(*
  Detects Marks and generates StartTrigger based on one EL1252 timestamp input I/O.
  Implements a CameraTrigger instance as well.
  
  Additionally:
    - returns lateral offset (+/- in [m]) to center of detected marks.
    - manages & supervises mark sequence
    - is a CameraTrigger as well
    - supports simulation mode
  
  NOTE: 
    - a mark has always a rising and falling edge of the sensor (triangle)
    - center position is the middle of the triangular mark

*)
FUNCTION_BLOCK FB_MarkDetection_v1 EXTENDS T_NamedBase IMPLEMENTS I_StartPosDetect, I_CameraTrigger, I_Sim
VAR_INPUT
  (*EL1252*)
  bIKp_StartSensor          AT%I* : BOOL;             (*Sensor start trigger*)
  tIKp_TimeStampPos         AT%I* : T_DCTIME64;       (*TimeStamp Pos_Edge @EL1252*)
  tIKn_TimeStampNeg         AT%I* : T_DCTIME64;       (*TimeStamp Neg_Edge @EL1252*)

  // configuration
  bEnable                         : BOOL;             (*Enable start pos detection sensor (from extern)*)
  bAutomaticMode                  : BOOL;             (*machine is in automatic mode *)
  nCurrentPos                     : DINT;             (*current position in Pulses/Subpixels*)
  fCurrentSpeed                   : LREAL;            (*actual speed of conveyor in [m/s]*)
  bReverse                        : BOOL;             (*reverse printing same roll feeded in opposite direction, check falling edge in this case*)
  
  // Debug & Test
  bManualTrigger                  : BOOL;             // Manual start trigger
  bManualReset                    : BOOL;             // Manaul reset detection
END_VAR
VAR
  bInitOk                         : BOOL;             // fb initialized

  // config
  _fResolution                    : LREAL := 1;       // current used print resolution (dpi*SubPx)
  _pFbMarkDefinition              : POINTER TO FB_MarkDefinition;      // mark definition
  _iCamera                        : I_Camera;         // camera interface
  // settings                                    
  _bUseCameraTrigger              : BOOL;             // (cam specific setting) Generate camera trigger output
  _bUseCameraTriggerFeedback      : BOOL;             // (cam specific setting) Evaluate camera triggered feedback
  _bCamManualTeachMode            : BOOL;             // cam in manual teach mode
  _fSubstrateLength               : LREAL;            // Substrate length in [m] (should be repeat ength)
  _fTriggerDistance               : LREAL;            // Distance between Sensor and Trigger [m]
  _fTriggerLength                 : LREAL := 10;      // Length of trigger signal in ms, min. 3 bus cycles
  _iActiveCam                     : I_CameraTriggerDevice;  // active camera interface (set by Enable() on I_CameraTrigger)

  // sensor
  bSheetActive                    : BOOL;             (*sheet is scanning*)
  bSpeedValid                     : BOOL;             (*speed is valid*)
  bTriggerArmed                   : BOOL;             (*trigger is armed*)
  bCamValid                       : BOOL;             (*camera is valid*)
  bMarkValid                      : BOOL;             (*definition is valid marks&substrate*)
  
  // helper
  rfT_Enable                      : RF_TRIG;          // edge detection enable
  bResetDetection                 : BOOL;             // Reset request for checkForMark() internals
  isStartMark                     : BOOL;
  isMarkError                     : BOOL;
  nMarkSelection                  : UDINT := 1;       // Current selected mask to search
  pMarkSearch                     : POINTER TO ST_MarkDefinition;
  _fSubstrateLengthEffective      : LREAL;            // Substrate length in [m]
  
  // time calculations
  tNowDc                          : T_DCTIME64;       // Get Current Timestamp (now)
  fCycleTime                      : LREAL;            // Current calculated cycle time [s]
  
  // I_StartPosDetect
  _bStartTrig                     : BOOL;             // Start Trigger Edge
  _nX0                            : DINT;             // X0 Position [SubPx]
  _bValid                         : BOOL;             //
  
  // simulation & debug
  _bSimEnable                     : BOOL;             // simulation mode enabled
  _bVerbose                       : BOOL;             // verbose mode
  _fSubstrateGap                  : LREAL;            // Gap between two substrates (sheets/repeats) for simulation
  
  // local for checkForMark
  rfEdgeSensor                    : RF_TRIG;          // edge detection start trigger
  tRisingEdge, tFallingEdge       : T_DCTIME64;       // detected edges
  nRisingPos, nFallingPos         : DINT;             // detected [SubPx] pos
  fMarkDuration                   : LREAL;            // duration in rising-falling time delta
  nLastStartMarkPosition          : DINT;             // last detected start mark
  bMarkStartDetected              : BOOL;             // mark started
  bMarkEndDetected                : BOOL;             // marks end reached
  
  bInhibitTrigger                 : BOOL;             // inhibit sensor signals, TRUE=inhibit
  
  // history 
  // - repeat
  sRepeatHistory : ARRAY[0..nC_HistorySize-1] OF ST_RepeatHistory;   // detection history
  nRepeatCt : UDINT;                 // history entry selector
  // flags for reapeat history
  bLenNotInRange_Repeat  : BOOL;     // Effective length not in range
  bStartOverrun_Repeat   : BOOL;     // too many starts
  bMissingMarks_Repeat   : BOOL;     // ...
  bMarksTooShort_Repeat  : BOOL;     // ...
  bMarksDetectErr_Repeat : BOOL;     // ...
  // - marks
  sMarkHistory : ARRAY[0..nC_HistorySize-1] OF ST_MarkDefinition;   // history of detected marks
  nMarkHistoryCt : UDINT;            // history entry selector
  // simulation
  bSim_Mark_Dev : BOOL;
  fSim_Mark_DevX, fSim_Mark_DevY : LREAL;     // simulate some fix deviation of detected marks [m]
END_VAR
VAR PERSISTENT
  bR_TerminateLast                : BOOL;             // Terminate sheet with last defined & detected mark
  nR_SpeedMavFilterSamples        : UINT := 0;        // moving average filter samples = 0 deactivated
END_VAR
VAR CONSTANT
  fC_MinimalSpeed                 : LREAL := 0.010;   // [m/s] speed valid (used for trigger activation)
  fC_MarkLengthMargin             : LREAL := 0.005;   // [m] used for mark end position supervision (mark end missed)
  fC_MaxSubstrateFactor           : LREAL := 1.1;     // factor which the sheet length can be max. longer
  nC_AreaMarkSensorOk             : INT := 10;        // [%] Area with the correct arrangement of the mark sensor
  nC_HistorySize                  : UDINT := 20;
END_VAR

// check parameter
IF NOT bInitOk THEN RETURN; END_IF

// General calculations
bSpeedValid   := fCurrentSpeed > fC_MinimalSpeed;                // speed valid (ignore trigger if not moving)
bCamValid     := SEL(_iActiveCam<>0, FALSE, TRUE);               // camera valid (ignore trigger otherwise)
bMarkValid    := (_fSubstrateLength > 0 AND _pFbMarkDefinition^.nMarks > 0);
tNowDc        := F_GetCurDcTaskTime64();                         // current dc time (most accurate time stamp we have)
fCycleTime    := calcCycleTime(tCurrent:=tNowDc);                // calculate cycle time of this fb
bTriggerArmed :=  bCamValid AND bSpeedValid AND bEnable AND bMarkValid AND (bAutomaticMode OR _bCamManualTeachMode OR _bSimEnable);   // trigger

IF bCamValid THEN    // (not yet used) save dynamic changable settings
  _fTriggerDistance := _iActiveCam.fTriggerDistance;
  _fTriggerLength   := _iActiveCam.fTriggerPulseLength;
END_IF

_bValid := _bStartTrig := FALSE;    // default values (outputs and properties)

manualTrigger();     // handle manual trigger


// enable & reset
rfT_Enable(CLK:=bEnable);             // edge detection (or use bTriggerArmed)
IF rfT_Enable.RT OR rfT_Enable.FT OR bManualReset THEN Reset(); bManualReset:=FALSE; END_IF;
IF NOT bEnable THEN RETURN; END_IF    // do nothing if not enabled
IF NOT bTriggerArmed THEN RETURN; END_IF


// Work
// - detect marks
//   - detect missing marks (based on teach definition, type and a margin)
//   - maybe replace missing marks (trend or teach)
// - handle StartTrigger if StartMark rising edge
// - handle Mark detected position (y-correction)
// - save mark, keep tracking of detected marks, (error handling if some missed)
// - send mark to camera


(*State Machine ----------------------------------------------------------------*)
// select mark
IF nMarkSelection > _pFbMarkDefinition^.nMarks THEN nMarkSelection := 1; END_IF  // fix invalid selection
pMarkSearch :=  _pFbMarkDefinition^.getMark(nIdx:=TO_DINT(nMarkSelection));

// search for mark
IF checkForMark(pMark:=pMarkSearch, bStartMark=>isStartMark, bErr=>isMarkError) THEN 

  IF _bVerbose THEN LogInfo(F_Concat4('found ', SEL(isStartMark,'Intermediate','StartMark'), SEL(isMarkError,' OK ',' ERR '), strMark(pMark:=pMarkSearch))); END_IF  

  // searched start, found start (normal start)
  IF isStartMark AND nMarkSelection = 1 THEN
    IF _pFbMarkDefinition^.nMarks = 1 THEN 
      // only one mark --> TERMINATE + START
      // - start
      SheetStart(pMark:=pMarkSearch);
      IF bR_TerminateLast THEN SheetStop(nNewX0:=0); END_IF  // TERMINATE already after single mark scanned
    ELSE
      // more marks --> START + NEXT
      // - start
      SheetStart(pMark:=pMarkSearch);
      // - next
      nMarkSelection := nMarkSelection + 1;    // next mark
		END_IF

  // search other mark and found start mark (start abort)
  ELSIF isStartMark AND nMarkSelection > 1 THEN
    // terminate(abort) last
    IF nMarkSelection < _pFbMarkDefinition^.nMarks THEN
      LogError('New start mark before last mark detected, missed a mark?');
      bMissingMarks_Repeat := TRUE;
    END_IF

    // terminate/abort with new --> TERMINATE + START
    // - start
    SheetStart(pMark:=pMarkSearch);
    
    nMarkSelection := nMarkSelection + 1;    // next mark

  // intermediate marks
  ELSIF NOT isStartMark AND nMarkSelection > 1 THEN
    // search and found other --> NEXT (ev. terminate)
    
    IF _pFbMarkDefinition^.nMarksDetected <= _pFbMarkDefinition^.nMarks THEN
      // - save mark
        _pFbMarkDefinition^.saveMark(pMark:=pMarkSearch);   // save
      // - last mark?
      IF nMarkSelection = _pFbMarkDefinition^.nMarks THEN
        IF bR_TerminateLast THEN SheetStop(nNewX0:=0); END_IF   // stop ct
        nMarkSelection := 1;
      ELSE
        nMarkSelection := SEL(nMarkSelection<_pFbMarkDefinition^.nMarks, 1, nMarkSelection + 1);  // next
      END_IF 
    END_IF
	END_IF
  
END_IF



// outputs
// _bStartTrig := // set in SheetStart
// _nX0 :=  // set in SheetStart
_bValid := TRUE;

(*
  Check if mark was detected properly and type matches.
  :returns:  TRUE if valid mark
*)
METHOD PRIVATE analizeMark : BOOL
VAR_INPUT
  pMark           : POINTER TO ST_MarkDefinition;     // mark to search for
  nDetectedPos    : DINT;                             // detected position [SubPx]
  fRealMarkLength : LREAL;                            // real detected mark length [m]
END_VAR
VAR_OUTPUT
  bStartMark : BOOL;    // a start mark was detected
  bTooLong : BOOL;      // detected length was too short for given mark
  bTooShort : BOOL;     // detected length was too long for given mark
END_VAR
VAR
  fMarkLengthMin : LREAL;
  fMarkLengthMax : LREAL;
END_VAR
IF pMark = 0 THEN RETURN; END_IF
IF pMark^.fHeight = 0 OR pMark^.fTrLength = 0 THEN analizeMark := FALSE; RETURN; END_IF
(*
  Sensor should aligned to the middle of the sensor (fI_MarkHeight / 2)
  With the difference OF the measured length to the normal lenght, the LateralOffset in Y can be calculated
*)

pMark^.sState.nPosXReal := nDetectedPos;          // save detected mark pos (rising in normal, falling in reverse print)
pMark^.sState.fLengthReal := fRealMarkLength;     // apply detected mark length

fMarkLengthMin := pMark^.fSqLength;
fMarkLengthMax := pMark^.fSqLength+pMark^.fTrLength;
// - minimal mark length check
IF fRealMarkLength < fMarkLengthMin THEN
  // mark shorter than defined, ignore detected
  //LogError(F_Concat6('Mark[', TO_STRING(pMark^.nId) ,'] too short ', TO_STRING(fRealMarkLength), '<', TO_STRING(fMarkLengthMin)));
  bTooShort := TRUE;
  RETURN; 
END_IF
// - max mark length check
IF fRealMarkLength > (_pFbMarkDefinition^.fMaxLengthStartMark + fC_MarkLengthMargin) THEN
  // mark even longer than longer max size of StartMark
  //LogError(F_Concat4('Mark too long ', TO_STRING(fRealMarkLength), '>', TO_STRING(fMarkLengthMax)));
  bTooLong := TRUE; 
RETURN; END_IF 

// - dx  (based on sheet begin) dx = current mark position - teached mark position
IF NOT bSim_Mark_Dev THEN pMark^.sState.dx := getMarkDistanceEffective(pMark:=pMark) - pMark^.fPosX;
ELSE                      pMark^.sState.dx := fSim_Mark_DevX;
END_IF

// - dy
IF NOT bSim_Mark_Dev THEN pMark^.sState.dy := ((pMark^.sState.fLengthReal - pMark^.fSqLength)/pMark^.fTrLength)*pMark^.fHeight-(pMark^.fHeight/2);
ELSE                      pMark^.sState.dy := fSim_Mark_DevY;
END_IF
IF pMark^.bInvertedX THEN     // if marks are inverted (flipped along x-axis), the correction is inverted
  pMark^.sState.dy := -1*pMark^.sState.dy;
END_IF

// check position qualitiy
pMark^.sState.bInArea := FC_COMPARE_RANGE_PERCENT( 
                                       fI_ValueSet := (pMark^.fHeight / 2)
                                     , fI_ValueActual  := (pMark^.fHeight / 2) + pMark^.sState.dy
                                     , fI_RangePercent := nC_AreaMarkSensorOk);

// type of mark
bStartMark := (fRealMarkLength >= _pFbMarkDefinition^.fMinLengthStartMark);
pMark^.sState.bSet := TRUE;

analizeMark := pMark^.sState.bSet;
END_METHOD

PROPERTY bManualTeach : BOOL
GET
bManualTeach := _bCamManualTeachMode;
END_GET
SET
_bCamManualTeachMode := bManualTeach;
END_SET
END_PROPERTY

{attribute 'monitoring' := 'call'}
(*Simulation is enabled set/get*)
PROPERTY bSimEnable : BOOL
GET
bSimEnable := _bSimEnable;
END_GET
SET
_bSimEnable := bSimEnable;
END_SET
END_PROPERTY

(*
  A new container detected.
  NOTE: a pulse only
*)
PROPERTY bStartTrig : BOOL
GET
bStartTrig := _bStartTrig;
END_GET
END_PROPERTY

(*
  A valid container detected.
*)
PROPERTY bValid : BOOL
GET
bValid := _bValid;
END_GET
END_PROPERTY

// cycle time in [s]
METHOD PRIVATE calcCycleTime : LREAL
VAR_INPUT
  tCurrent : T_DCTIME64;
END_VAR
VAR_INST
  tLastTimeStamp : T_DCTIME64 := 0;
END_VAR
calcCycleTime := (TO_LREAL(tCurrent) - TO_LREAL(tLastTimeStamp)) * 1E-9;
tLastTimeStamp  := tCurrent;  // memory timestamp
END_METHOD

(*
  Poll for sensor triggers and marks.
  :return: true if a mark was detected
*)
METHOD PRIVATE checkForMark : BOOL
VAR_INPUT
  pMark : POINTER TO ST_MarkDefinition;             // mark to search for
END_VAR
VAR_OUTPUT
  bErr : BOOL;                // 
  bStartMark : BOOL;          // a start mark was detected
END_VAR
VAR
  nAbortMarkAfter : DINT;     // max. length to search for mark end before aborting this mark [SubPx]
  bTooShort, bTooLong : BOOL;
END_VAR
IF pMark = 0 THEN RETURN; END_IF
IF bResetDetection THEN   // reset methods internal states
  bMarkStartDetected := FALSE; bMarkEndDetected := FALSE;
  bInhibitTrigger := FALSE; 
  bResetDetection := FALSE;
  bErr := FALSE;
END_IF

// --- Simulation for testing
IF _bSimEnable THEN   // simulate some marks for testing
  checkForMark := SimMarks(pMark:=pMark, bStartMark=>bStartMark);
  RETURN; 
  
// --- Generate masks if none are available
ELSIF pMark^.bVirtual THEN    // generate marks (for NoMark mode)
  checkForMark := GenMark(pMark:=pMark, bStartMark=>bStartMark);
  RETURN;
END_IF


// --- Use sensor
rfEdgeSensor(CLK:=bIKp_StartSensor);   // edge detection
nAbortMarkAfter := F_MeterToSubPixel(fPosMeter:=pMark^.fTrLength + pMark^.fSqLength + fC_MarkLengthMargin + fCycleTime*fCurrentSpeed, fResoSubPx:=_fResolution); // mark len + margin + one cycle

// -- rising edge detection
IF rfEdgeSensor.RT AND NOT bInhibitTrigger THEN
  tRisingEdge := tIKp_TimeStampPos;   // sample input
  nRisingPos  := getExactPosition(tNow:=tNowDc, tEdge:=tRisingEdge, nPos:=nCurrentPos, fSpeed:=fCurrentSpeed);   // position where mark was seen
  bMarkStartDetected := TRUE;
END_IF;
// -- falling edge detection
IF rfEdgeSensor.FT AND NOT bInhibitTrigger THEN
  // falling edge
  tFallingEdge := tIKn_TimeStampNeg;
  nFallingPos := getExactPosition(tNow:=tNowDc, tEdge:=tFallingEdge, nPos:=nCurrentPos, fSpeed:=fCurrentSpeed);   // position where mark was seen
  IF NOT bMarkStartDetected THEN
    // abort
    bErr := TRUE; LogError('Missing rising trigger edge before falling edge');
    bMarksDetectErr_Repeat := TRUE;
  ELSE
    // ok                    
    bMarkEndDetected := TRUE; 
  END_IF
END_IF
// - abort search for end
IF bMarkStartDetected AND (nCurrentPos - nRisingPos) > nAbortMarkAfter THEN      // abort after waiting for end
  // Abort - Expected falling edge missed
  bErr := TRUE; LogWarning(F_Concat2('Mark end not given after [SubPx]:', TO_STRING(nAbortMarkAfter)));
  bMarksDetectErr_Repeat := TRUE;
  //  nFallingPos := nRisingPos + F_MeterToSubPixel(fPosMeter:=pMark^.fTrLength/2+pMark^.fSqLength, fResoSubPx:=_fResolution);  // set still a valid pos
  //  bMarkEndDetected := TRUE;
  //  pMark^.sState.bMissed := TRUE;
END_IF;

// mark evaluation 
IF bMarkStartDetected AND bMarkEndDetected THEN
 
  // check mark & calculate offsets
  fMarkDuration := ABS(ULINT_TO_LREAL(tFallingEdge) - ULINT_TO_LREAL(tRisingEdge));		// Calculate how long the signal was ON
  // define and check mark
  IF analizeMark( pMark:=pMark,
                  nDetectedPos:=SEL(bReverse, nRisingPos, nFallingPos),
                  fRealMarkLength:=fMarkDuration * fCurrentSpeed * 0.000_000_001,
                  bStartMark => bStartMark,
                  bTooLong => bTooLong,
                  bTooShort => bTooShort,
               )
  THEN
    checkForMark := TRUE;      // a valid mark detected
  ELSE
    IF bTooShort THEN bMarksTooShort_Repeat := TRUE; bMarksDetectErr_Repeat := TRUE; END_IF   // apply some error tracing
    IF bTooLong THEN bMarksDetectErr_Repeat := TRUE; END_IF   // apply some error tracing
    bErr := TRUE;  // invalid mark detected
	END_IF
  
 
  SaveToMarkHistory(pMark:=pMark);    // Save to mark history
  
  bResetDetection := TRUE;   // reset detection logic
END_IF

IF bErr THEN bResetDetection := TRUE; END_IF    // reset marks on any error as well
END_METHOD

METHOD Disable : BOOL
_iActiveCam := 0;
Disable := TRUE;
END_METHOD

METHOD Enable : BOOL
VAR_INPUT
	iCam	                    : I_CameraTriggerDevice;
  bUseCameraTrigger         : BOOL; //Generate camera trigger
  bUseCameraTriggerFeedback : BOOL; //Use feedback as trigger?
END_VAR
IF iCam = 0 THEN
  Enable := FALSE;
  LogError('setCam failed: invalid reference');
ELSE
  _iActiveCam := iCam;
  Enable     := TRUE;

  // save constant settings
  _bUseCameraTrigger := bUseCameraTrigger;
  _bUseCameraTriggerFeedback := bUseCameraTriggerFeedback;
  
  IF _bUseCameraTrigger OR _bUseCameraTriggerFeedback THEN
    LogWarning('Enable: Camera Trigger output/feedback not yet supported');
	END_IF
END_IF;
END_METHOD

PROPERTY fSubstrateGap : LREAL
SET
_fSubstrateGap := fSubstrateGap;
END_SET
END_PROPERTY

(*
  Generate detected marks.
*)
METHOD PRIVATE GenMark : BOOL
VAR_INPUT
  pMark : POINTER TO ST_MarkDefinition;
END_VAR
VAR_OUTPUT
  bStartMark : BOOL;
END_VAR
VAR_INST
  bMarkOn : BOOL;
  n : DINT;
  nImageLength : DINT;
END_VAR
IF pMark = 0 THEN RETURN; END_IF

nImageLength := F_MeterToSubPixel(fPosMeter:=_fSubstrateLength + _fSubstrateGap, fResoSubPx:=_fResolution);
IF nImageLength = 0 THEN RETURN; END_IF


IF NOT bMarkOn THEN  // start new mark

  // create rising edge
  IF pMark^.nId = 1 THEN          // a start mark
    // wait for next StartPosition
    IF nCurrentPos >= nLastStartMarkPosition + nImageLength THEN

      // fix bigger gaps than next sheet (always try to start repeats at a multiple of last repeat)
      IF (nCurrentPos - nLastStartMarkPosition) / nImageLength > 2 THEN
        nLastStartMarkPosition := nLastStartMarkPosition + ((((nCurrentPos - nLastStartMarkPosition) / nImageLength) -1) * nImageLength);  // correct to one sheet before 
			END_IF 
      
      nLastStartMarkPosition := nLastStartMarkPosition + nImageLength;      // save last repeat position   
      
      pMark^.sState.nPosXReal := nLastStartMarkPosition + F_MeterToSubPixel(fPosMeter:=pMark^.fPosX, fResoSubPx:=_fResolution); // mark detected position
      pMark^.sState.fLengthReal := 0;
      pMark^.sState.dx := 0;
      pMark^.sState.dy := 0;
      pMark^.sState.bInArea := TRUE;
      pMark^.sState.bSet := TRUE;
      bMarkOn := TRUE;
    END_IF
	ELSE
    // wait for next mark position
    IF F_SubPixelToMeter(lPosSubPx:=ABS(nCurrentPos - nLastStartMarkPosition), fResSubPx:=_fResolution) >= pMark^.fPosX THEN
     
      pMark^.sState.nPosXReal := nLastStartMarkPosition + F_MeterToSubPixel(fPosMeter:=pMark^.fPosX, fResoSubPx:=_fResolution); // 
      pMark^.sState.fLengthReal := 0;
      pMark^.sState.dx := 0;
      pMark^.sState.dy := 0;
      pMark^.sState.bInArea := TRUE;
      pMark^.sState.bSet := TRUE;
      bMarkOn := TRUE;
		END_IF
  END_IF
  
ELSE
  // end mark after one dycle
  bMarkOn := FALSE;
  IF pMark^.nId = 1 THEN bStartMark := TRUE; END_IF  
  GenMark := TRUE;      // reset after one cycle active
  SaveToMarkHistory(pMark:=pMark);    // Save to mark history
END_IF
END_METHOD

// calculate the exact detected position
// :returns: the X0 position
METHOD PRIVATE getExactPosition : DINT
VAR_INPUT
  tNow : T_DCTIME64;    // current system time
  tEdge : T_DCTIME64;   // detected time
  nPos : DINT;          // current (encoder) position at the current time
  fSpeed : LREAL;       // current speed for the timestamped position correction calculation
END_VAR
VAR
  fDeltaDistance : LREAL;       // Distance that the substrate moved between the detection and the treatment of the information
END_VAR
// calculation like DMAX
fDeltaDistance := UINT64_TO_LREAL(UInt64Sub64(ULINT_TO_ULARGE(tNowDc), ULINT_TO_ULARGE(tEdge))) * 1E-9 * fSpeed;
getExactPosition := nPos - TO_DINT(fDeltaDistance); 

// before calculation with some compensation
(*
  // Calculate the original position in our position domain
  tCurrentTime  := F_GetCurDcTaskTime64();
  fL_CurrentTimeStamp  := (ULINT_TO_LREAL(tCurrentTime) - (nC_CurrentTimeStampComp * 1_000)) / 1_000_000.0; (*in ms*)
  fI_Sensor_TimeStamp := (ULINT_TO_LREAL(tRisingEdge) - (nC_SensorTimeStampComp  * 1_000)) / 1_000_000.0; (*in ms*)

  // Treatment of the information
  fDeltaDistance := (fL_CurrentTimeStamp - fI_Sensor_TimeStamp) * 0.001 * fCurrentSpeed;	(* Distance in pulses that the substrate has traveled between the sensor detection and the PLC treatment *)
  iL_DeltaPosition := FC_LREAL_TO_DINT(fDeltaDistance * (1 / (0.0254 / fI_Resolution)));  (*1/1px*)	(* Travel of the substrate between the time of acquisition and the time of treatment *)
  nOffset_X0       := nCurrentPos - iL_DeltaPosition;	(* Position where the sheet has been detected *)
*)
END_METHOD

(*
  Get X0 from detected start mark
*)
METHOD PRIVATE getLastX0 : DINT
VAR
  pLastStartMark : POINTER TO ST_MarkDefinition;
END_VAR
pLastStartMark := _pFbMarkDefinition^.pLastStartMark;
IF pLastStartMark <> 0 THEN
  getLastX0 := pLastStartMark^.sState.nPosXReal - F_MeterToSubPixel(fPosMeter:=pLastStartMark^.fPosX, fResoSubPx:=_fResolution);
END_IF
END_METHOD

(*
  Calculate effective distance of mark to X0 [m]
*)
METHOD PRIVATE getMarkDistanceEffective : LREAL
VAR_INPUT
  pMark : POINTER TO ST_MarkDefinition;
END_VAR
VAR
  pFirstMark : POINTER TO ST_MarkDefinition;
END_VAR
IF pMark = 0 THEN RETURN; END_IF

IF pMark^.nId = 1 THEN 
  getMarkDistanceEffective := pMark^.fPosX;
ELSE
  pFirstMark := _pFbMarkDefinition^.getMark(nIdx:=1);
  IF pFirstMark <> 0 THEN
    // real distance between this mark and start mark + fPosX of start mark
    getMarkDistanceEffective := pFirstMark^.fPosX + F_SubPixelToMeter(lPosSubPx:=pMark^.sState.nPosXReal - pFirstMark^.sState.nPosXReal, fResSubPx:=_fResolution);
  END_IF
END_IF
END_METHOD

METHOD Init
VAR_INPUT
  fPrintResolution      : LREAL := 600;         // print(head) resolution in [dpi]
  fSubPxResolution      : LREAL := 32;          // SubPixel resolution [SubPx], resolution factor (fI_PrintResolution*fI_SubPxResolution=>Output resolution)
  pFbMarkDefinition     : POINTER TO FB_MarkDefinition;
END_VAR
VAR
  i : UDINT;
END_VAR
IF fPrintResolution = 0 OR fSubPxResolution = 0 OR pFbMarkDefinition = 0 THEN LogError('Init: invalid parameter'); RETURN; END_IF

_fResolution := fPrintResolution * fSubPxResolution;
_pFbMarkDefinition:= pFbMarkDefinition;

Reset();

bInitOk := TRUE;
END_METHOD

METHOD PRIVATE manualTrigger : BOOL
VAR_INST
  rfTrig_ManuTrigger : RF_TRIG;
END_VAR
rfTrig_ManuTrigger(CLK:=bManualTrigger);

IF rfTrig_ManuTrigger.RT THEN
  LogWarning('manualTrigger not yet implemented');
END_IF

manualTrigger := rfTrig_ManuTrigger.RT;
END_METHOD

(*
  Detected start position X0 (absolute) in [SubPx].
*)
PROPERTY nStartPositionX0 : DINT
GET
nStartPositionX0 := _nX0;
END_GET
END_PROPERTY

(*
  Reset internal state and all marks
*)
METHOD Reset
IF NOT bInitOk THEN RETURN; END_IF

_bValid := FALSE;
_bStartTrig := FALSE;
nMarkSelection := 1; // start mark

// reset camera (release if one is selected)
IF bSheetActive THEN
  IF _iActiveCam <> 0 THEN _iActiveCam.CamTriggerDone(); END_IF   // notify an done/abort
END_IF
_pFbMarkDefinition^.ResetMarkStates();  // reset detected marks
bSheetActive := FALSE;
bResetDetection := TRUE;        // reset checkForMark() state machine
END_METHOD

METHOD PRIVATE SaveToMarkHistory
VAR_INPUT
  pMark : POINTER TO ST_MarkDefinition;
END_VAR
VAR
  i : UDINT;
END_VAR
FOR i:=0 TO nC_HistorySize-1 DO sMarkHistory[i].sView.colorFill := 16#FFE2DDDB; END_FOR   // clear selection
nMarkHistoryCt := (nMarkHistoryCt + 1) MOD nC_HistorySize;
sMarkHistory[nMarkHistoryCt] := pMark^;
sMarkHistory[nMarkHistoryCt].sView.colorFill := 16#FF90EE90;
END_METHOD

METHOD SetSubstrateLength
VAR_INPUT
  fSubstrateLength : LREAL;
END_VAR
IF NOT bInitOk THEN RETURN;END_IF;

(*reduced by margin (for endless mode with potential smaller printed repetition)*)
_fSubstrateLength := fSubstrateLength;
//_nSubstrateLength := F_MeterToSubPixel(fPosMeter:=_fSubstrateLength, fResoSubPx:=_fResolution);
END_METHOD

METHOD PRIVATE SheetStart
VAR_INPUT
  pMark : POINTER TO ST_MarkDefinition;
END_VAR
VAR
  sMarkBackup : ST_MarkDefinition;
END_VAR
_nX0 := pMark^.sState.nPosXReal - F_MeterToSubPixel(fPosMeter:=pMark^.fPosX, fResoSubPx:=_fResolution);
_bStartTrig := TRUE;

// (force) terminate a sheet/repeat
IF bSheetActive THEN 
  IF _bVerbose THEN LogInfo(F_Concat2('Terminate sheet/repeat with new Start Mark', '')); END_IF
  sMarkBackup := pMark^;   // push 
  SheetStop(nNewX0:=_nX0);
  pMark^:= sMarkBackup;    // pop
END_IF

IF _bVerbose THEN LogInfo(F_Concat2('SheetStart at X0=', TO_STRING(_nX0))); END_IF

// save (start) mark
_pFbMarkDefinition^.saveMark(pMark:=pMark);

// trigger camera
IF _iActiveCam<>0 THEN _iActiveCam.CamTrigger(bOk:=TRUE, nPos:=_nX0, nPosDeviation:=0, nX0:=_nX0); END_IF

// reset debug states
bLenNotInRange_Repeat  := FALSE;
bStartOverrun_Repeat   := FALSE;
bMissingMarks_Repeat   := FALSE;
bMarksTooShort_Repeat  := FALSE;
bMarksDetectErr_Repeat := FALSE;

bSheetActive := TRUE;
END_METHOD

METHOD PRIVATE SheetStop
VAR_INPUT
  nNewX0 : DINT;   // new detected X0
END_VAR
VAR
  i : UDINT;
  pLastMark : POINTER TO ST_MarkDefinition;
  fD : LREAL;
  fSLen : LREAL;
  nDetectedX0 : DINT;
END_VAR
// - terminate
IF _bVerbose THEN LogInfo(F_Concat2('SheetStop()', '')); END_IF

fSLen := _fSubstrateLength;  // (default) original length

// calculate effective sheet length
nDetectedX0 := getLastX0();   // get sampled X0
IF nNewX0 <> 0 AND nDetectedX0 <> 0 THEN
  // real diff between two starts
  fD := F_SubPixelToMeter(lPosSubPx:=nNewX0 - nDetectedX0, fResSubPx:=_fResolution);
  IF fD < (_fSubstrateLength * fC_MaxSubstrateFactor) THEN
    fSLen := fD;
  END_IF 
ELSIF nNewX0 = 0 AND _pFbMarkDefinition^.nMarksDetected > 1 THEN
  // calculate based on last detected mark (a strech factor)
  pLastMark:= _pFbMarkDefinition^.getMark(nIdx:=0);     // get last available mark
  fD := getMarkDistanceEffective(pMark:=pLastMark); 
  fSLen := (pLastMark^.fPosX/SEL(fD<>0, pLastMark^.fPosX, fD)) * _fSubstrateLength; // estimate real length with last mark
END_IF
_fSubstrateLengthEffective := fSLen;


// debug history
FOR i:=0 TO nC_HistorySize-1 DO sRepeatHistory[i].bSelected := FALSE; END_FOR   // clear selection
nRepeatCt := (nRepeatCt + 1) MOD nC_HistorySize;
sRepeatHistory[nRepeatCt].bSelected       := TRUE;
sRepeatHistory[nRepeatCt].nIndex          := nRepeatCt+1;
sRepeatHistory[nRepeatCt].nX0             := nDetectedX0;
sRepeatHistory[nRepeatCt].fLen            := _fSubstrateLength;
sRepeatHistory[nRepeatCt].fLenEffective   := _fSubstrateLengthEffective;
sRepeatHistory[nRepeatCt].fLenDiff        := _fSubstrateLengthEffective - _fSubstrateLength;
sRepeatHistory[nRepeatCt].bLenNotInRange  := bLenNotInRange_Repeat;
sRepeatHistory[nRepeatCt].bStartOverrun   := bStartOverrun_Repeat;
sRepeatHistory[nRepeatCt].bMissingMarks   := bMissingMarks_Repeat;
sRepeatHistory[nRepeatCt].bMarksTooShort  := bMarksTooShort_Repeat;
sRepeatHistory[nRepeatCt].bMarksDetectErr := bMarksDetectErr_Repeat;


IF _iActiveCam<>0 THEN _iActiveCam.CamTriggerDone(); END_IF 
_pFbMarkDefinition^.ResetMarkStates();

bSheetActive := FALSE;
END_METHOD

METHOD PRIVATE SimMarks : BOOL
VAR_INPUT
  pMark : POINTER TO ST_MarkDefinition;
END_VAR
VAR_OUTPUT
  bStartMark : BOOL;
END_VAR
VAR_INST
  bMarkOn : BOOL;
  nMarkStarted : DINT;
  fStartMarkOffset : LREAL;
  rand : DRAND;
  rlrand : LREAL;
  l : DINT;
END_VAR
IF pMark = 0 THEN RETURN; END_IF

// when sim enabled AND auto-trigger then create a StartMark after every sheet/repeat length
//  then generate every following intermediate mark with a given length

IF NOT bMarkOn THEN  // start new mark
  // create rising edge
  IF pMark^.nId = 1 THEN
    // wait for next StartPosition
    IF F_SubPixelToMeter(lPosSubPx:=ABS(nCurrentPos - nLastStartMarkPosition), fResSubPx:=_fResolution) >= _fSubstrateLength + _fSubstrateGap THEN
      nLastStartMarkPosition := nCurrentPos;      // save start mark pos
      fStartMarkOffset := pMark^.fPosX;   // save start mark displacement from X0
      pMark^.sState.nPosXReal := nCurrentPos;  // save rising edge
      nMarkStarted := nCurrentPos;
      l := F_MeterToSubPixel(fPosMeter:=pMark^.fSqLength + (pMark^.fTrLength/2), fResoSubPx:=_fResolution); // mark length
      bMarkOn := TRUE;
    END_IF
	ELSE
    // wait for next mark position
    IF F_SubPixelToMeter(lPosSubPx:=ABS(nCurrentPos - nLastStartMarkPosition), fResSubPx:=_fResolution) >= pMark^.fPosX - fStartMarkOffset THEN
      pMark^.sState.nPosXReal := nCurrentPos;  // save rising edge
      nMarkStarted := nCurrentPos;
      l := F_MeterToSubPixel(fPosMeter:=pMark^.fSqLength + (pMark^.fTrLength/2), fResoSubPx:=_fResolution); // mark length
      bMarkOn := TRUE;
		END_IF
  END_IF
  
ELSE
  // create falling edge
  IF (nCurrentPos - nMarkStarted) > l THEN
    rand(Seed:=13, Num=>rlrand);  // TODO: find a right scale 
    analizeMark(pMark:=pMark, nDetectedPos:=nMarkStarted, fRealMarkLength:=F_SubPixelToMeter(lPosSubPx:=nCurrentPos - nMarkStarted, fResSubPx:=_fResolution));
    bMarkOn := FALSE;
    If pMark^.nId = 1 THEN bStartMark := TRUE; END_IF
    SimMarks := TRUE;    // mark done
    SaveToMarkHistory(pMark:=pMark);    // Save to mark history
  END_IF
END_IF
END_METHOD

METHOD strMark : T_MaxString
VAR_INPUT
  pMark : POINTER TO ST_MarkDefinition;
END_VAR
VAR_INST
  fbStrFormat : FB_FormatString;
END_VAR
VAR
  IdFormatted : STRING;
END_VAR
fbStrFormat(sFormat:='%.2d', arg1:=F_DINT(pMark^.nId), sOut=>IdFormatted);
strMark := F_Concat6(
  F_Concat2('Id:',   IdFormatted),
  F_Concat2(' Set:', SEL(pMark^.sState.bSet,'0','1')),
  F_Concat2(' posX:', LREAL_TO_FMTSTR( pMark^.fPosX, 5, TRUE )),
  F_Concat2(' posY:', LREAL_TO_FMTSTR( pMark^.fPosY, 5, TRUE )),
  F_Concat2(' dx:', LREAL_TO_FMTSTR( pMark^.sState.dx, 5, TRUE )),
  F_Concat2(' dy:', LREAL_TO_FMTSTR( pMark^.sState.dy, 5, TRUE )),
);
END_METHOD

END_FUNCTION_BLOCK

(* stored: Version 1.1.0.1, ProductVersion 3.1.4024.11
   POU FB_MarkDetection_v1: Id {b62150a6-825e-437a-9373-f5f855e5f86e}, SpecialFunc None
   Folder I_CameraTrigger: Id {56180a19-3b15-4d81-8547-a0739ec5c7f3}
   Folder I_Sim: Id {5bf14578-1cd1-48e6-8ccb-a561e61fca37}
   Folder I_StartPosDetect: Id {d9ce600f-3b3c-4ad1-a039-17015f10f9a3}
   Folder Sim: Id {6e17e2ff-1307-4f1e-a7aa-0112b5f8c092}
   Method analizeMark: Id {0fe27d59-09a3-4778-96a6-e1374e41ae68}
   Property bManualTeach: Id {0394ea46-e479-4b01-8e40-b42e26976645}
   Get Get: Id {72d372fe-ffbd-4427-9a95-46d8b9f4cf62}
   Set Set: Id {cfb0ce6c-fda7-4d17-bec9-544c3d2295c8}
   Property bSimEnable: Id {114cef08-ef9f-4655-a24a-d26bd75bffc8}
   Get Get: Id {94150729-07d7-4688-bfab-b53e757cf52c}
   Set Set: Id {18420c6e-8cc0-4506-8392-c504c5539a93}
   Property bStartTrig: Id {54688268-75b4-4e54-adee-9ba78173fccb}
   Get Get: Id {2d46a272-6e9d-4a92-b0ef-f6884b3ac027}
   Property bValid: Id {80a104b8-edb3-4882-883b-4d217d37420c}
   Get Get: Id {4de03f0a-e748-4062-9ecc-49d0fbbb8769}
   Method calcCycleTime: Id {c5da9bc5-c89b-4d56-983b-87158bdbb28a}
   Method checkForMark: Id {5b5c61c6-faec-413a-b0fc-c62604001c4a}
   Method Disable: Id {568fbd66-37a4-4787-b6c9-f80109bbf4eb}
   Method Enable: Id {65ffe8ba-a2c4-457f-8248-f36c7b7604d9}
   Property fSubstrateGap: Id {aa4395c4-e40d-41ec-b458-3a1d1f63f3fa}
   Set Set: Id {25f8767a-6942-4ecd-9f3b-22822a4dff57}
   Method GenMark: Id {2f317964-7083-44aa-8e69-e459b32a4afb}
   Method getExactPosition: Id {caab2ebd-553a-4e49-935d-0b7b1e82d497}
   Method getLastX0: Id {33d2561b-84c1-4070-bee0-64f7122e7896}
   Method getMarkDistanceEffective: Id {1f1e47da-e7ba-4b9b-8bcd-9447d37a1890}
   Method Init: Id {8ef9a6c7-7c5d-4ecb-ab2d-81464dbe108a}
   Method manualTrigger: Id {3e3bbe90-afeb-485c-a531-49f417b7ea76}
   Property nStartPositionX0: Id {cf3a635f-a07b-40ee-94a9-e8f8c803e2e1}
   Get Get: Id {c6f571fc-fcad-4d32-a21b-e241f24f58eb}
   Method Reset: Id {41704a3d-1ee5-4523-bb36-536ca832b13d}
   Method SaveToMarkHistory: Id {d87f8cb3-416b-4daf-90f8-5d127f8bbf85}
   Method SetSubstrateLength: Id {85e40680-5de7-433a-81b1-59e81722652b}
   Method SheetStart: Id {25997832-7f0a-4a0e-bced-1962863c1d9b}
   Method SheetStop: Id {aa4bc7d7-6e77-4e6b-a690-9267a6518d8b}
   Method SimMarks: Id {f2bb41e7-9b52-430a-b163-0f707b6ca248}
   Method strMark: Id {e8dcc4db-58b5-4337-a3fd-a299a10d8a8a} *)
